PROGRAM MAIN
VAR
	DateTime_TEST : DateTime_TEST;
	HelperFunctions_TEST : ConvertAnyToString_TEST;
	DynamicStringBuffer_TEST : DynamicStringBuffer_TEST;
	TestWrapper : TestWrapper_NET();
END_VAR

TcUnit.RUN();

TestWrapper();

END_PROGRAM

(* stored: Version 1.1.0.1
   POU MAIN: Id {899b5391-5363-4fd8-835e-d1662fef51af}, SpecialFunc None *)
